(* PLC project SafeLOGIC-1, BrAutomation SafeDESIGNER  4.4.0.0 *)
(* stored: companyURL http://www.br-automation.com, creationDateTime Mon May 10 15:18:38 2021 *)

PROGRAM Main

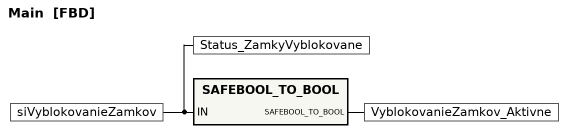
(* FBD diagram, written out as Structured Text *)
Status_ZamkyVyblokovane := siVyblokovanieZamkov;
VyblokovanieZamkov_Aktivne := SAFEBOOL_TO_BOOL(siVyblokovanieZamkov);
END_PROGRAM
